// TIA Portal V19 export
DATA_BLOCK "DB_Panel_Posinfo"   // DB52
{ S7_Optimized_Access := 'FALSE' }
// stored: AutoNumber false
   VAR RETAIN
      Offset : Int := 50;   // * Beginn Daten
      Leng : Int := 80;   // * Länge Daten
      resDW1 : DWord := 16#0000_0000;
      resDW2 : DWord := 16#0000_0000;
      resDW3 : DWord := 16#0000_0000;
      resDW4 : DWord := 16#0000_0000;
      last_Takt : DInt := 0;
      Taktzeit : DInt := 0;   // Zeit die der Takt läuft
      Takt_Ware : DInt := 0;   // Zeit seit Ausfahrt letzte Fertigware
      Stop_Anlage : Byte := 16#00;   // ungleich 0-->Kettenbearbeitung anhalten
      Feierabend : Byte := 16#00;   // ungleich 0-->FEIERABENDPROGRAMM
      Sonder_BA : Byte := 16#00;   // ungleich 0-->ELEKTROLYSE, ENTMETALLISIEREN
      IST_Sonder_BA : Byte := 16#00;
      FB_FW_akt : Word := 16#0000;   // an Fernbedienung gewählter FW
      SPS_getaktet : Bool := TRUE;
      resDW10 : DWord := 16#0000_0000;
      resDW11 : DWord := 16#0000_0000;
      resW : Word := 16#0000;
      Pos : Array[1..30] of Struct   // * Feldlänge anpassen
         Prio_Pos : Byte;   // Priorität des Bades (höchste Priorität==0
         lngsm_IN : Bool;   // langsames Einsetzen erforderlich-abhängig von immer_schnell
         lngsm_OUT : Bool;   // langsames Ausheben erforderlich-abhängig von immer_schnell
         res : Bool;
         res1 : Bool;
         res2 : Bool;
         res3 : Bool;
         Luft_Ein : Bool;   // Lufteinblasung ein
         Luft_Auto : Bool;   // Lufteinblasung Automatik
         Verweilzeit : DInt;   // Verweilzeit
         KF_A : Real;   // Korrekturfaktor WT_Auslastung 0..100%-->0..1, Gesamtoberfläche
         KF_Expo : Real;   // Korrekturfaktor Expozeit in %
         T_Vorruf : Int;   // Vorrufzeit lößt Vorruf n Sekunden vor Ablauf der Expozeit aus
         T_Pend : Int;   // Auspendelzeit 0..999s
         T_ATZ : Int;   // Abtropfzeit 0..999s
         NS_Auto : Bool;   // Nachspeisung Automatik
         SR_Auto : Bool;   // Spritzregister Automatik
         res6 : Bool;
         WBE_Ein : Bool;   // Warenbewegung ein
         WBE_Auto : Bool;   // Warenbewegung Automatik
         TS_Pos : Bool;   // Tropfschalenpos.
         res9 : Bool;
         res10 : Bool;
         resB : Byte;
         Niv_SPR : Int;   // Stärke Spritzen
         Zeit_SPR : Int;   // Zeit Spritzen
         Niv_Luft : Int;   // Stärke Lufteinblasung
         Zeit_Luft : Int;   // Zeit Lufteinblasung
         Niv_NS : Int;   // Niveau Füllstand in %
         Zeit_NS : Int;   // Nachspeisezeit getaktete NS
         NS_Kor_Tr : Byte;   // Korrektur Nachspeisezeit für Trommel
         Coun_Kor : Byte;   // Counter Korrektur Nachspeisung
         resD : DInt;
         resR_1 : Real;
         resR_2 : Real;
         resR_3 : Real;
         resI_1 : Int;
         resI_2 : Int;
         ExpoTol : DInt;   // Toleranz Expozeit
         SonDW1 : DInt;   // freie Nutzung Gesamtzeit Rüttler
         SonDW2 : DInt;   // freie Nutzung Intervall ein Rüttler
         SonDW3 : DInt;   // freie Nutzung Intervall aus Rüttler
         SonDW4 : DInt;   // freie Nutzung (Verzögerung US-Rüttler)
         T_Zt_SR : Int;   // Test-Zeit Spritzregister
         T_Zt_NS : Int;   // Test-Zeit Nachspeisung
      END_STRUCT;
   END_VAR
BEGIN
   Pos[1..9].Prio_Pos := 16#05;
   Pos[10].Prio_Pos := 16#00;
   Pos[11..12].Prio_Pos := 16#01;
   Pos[13..14].Prio_Pos := 16#00;
   Pos[15..16].Prio_Pos := 16#01;
   Pos[17].Prio_Pos := 16#00;
   Pos[18].Prio_Pos := 16#01;
   Pos[19].Prio_Pos := 16#00;
   Pos[20..21].Prio_Pos := 16#01;
   Pos[22].Prio_Pos := 16#00;
   Pos[23].Prio_Pos := 16#02;
   Pos[24..27].Prio_Pos := 16#05;
   Pos[28].Prio_Pos := 16#02;
   Pos[29].Prio_Pos := 16#03;
   Pos[30].Prio_Pos := 16#02;
   Pos[1..30].lngsm_IN := FALSE;
   Pos[1..30].lngsm_OUT := FALSE;
   Pos[1..30].res := FALSE;
   Pos[1..30].res1 := FALSE;
   Pos[1..30].res2 := FALSE;
   Pos[1..30].res3 := FALSE;
   Pos[1..30].Luft_Ein := FALSE;
   Pos[1..30].Luft_Auto := FALSE;
   Pos[1].Verweilzeit := 0;
   Pos[2].Verweilzeit := 2107;
   Pos[3].Verweilzeit := 2074;
   Pos[4].Verweilzeit := 0;
   Pos[5].Verweilzeit := 32100;
   Pos[6..7].Verweilzeit := 0;
   Pos[8].Verweilzeit := 115;
   Pos[9..23].Verweilzeit := 0;
   Pos[24].Verweilzeit := 300;
   Pos[25..27].Verweilzeit := 0;
   Pos[28].Verweilzeit := 32;
   Pos[29].Verweilzeit := 1;
   Pos[30].Verweilzeit := 0;
   Pos[1..30].KF_A := 1000.0;
   Pos[1..30].KF_Expo := 1.0;
   Pos[1..30].T_Vorruf := 0;
   Pos[1..30].T_Pend := 1;
   Pos[1..2].T_ATZ := 0;
   Pos[3..7].T_ATZ := 10;
   Pos[8..9].T_ATZ := 5;
   Pos[10].T_ATZ := 10;
   Pos[11..12].T_ATZ := 5;
   Pos[13..14].T_ATZ := 10;
   Pos[15..16].T_ATZ := 5;
   Pos[17].T_ATZ := 10;
   Pos[18].T_ATZ := 5;
   Pos[19].T_ATZ := 10;
   Pos[20..21].T_ATZ := 5;
   Pos[22].T_ATZ := 10;
   Pos[23].T_ATZ := 5;
   Pos[24..27].T_ATZ := 2;
   Pos[28].T_ATZ := 0;
   Pos[29].T_ATZ := 5;
   Pos[30].T_ATZ := 2;
   Pos[1..30].NS_Auto := FALSE;
   Pos[1..25].SR_Auto := FALSE;
   Pos[26].SR_Auto := TRUE;
   Pos[27..29].SR_Auto := FALSE;
   Pos[30].SR_Auto := TRUE;
   Pos[1..30].res6 := FALSE;
   Pos[1..30].WBE_Ein := FALSE;
   Pos[1..30].WBE_Auto := FALSE;
   Pos[1..30].TS_Pos := FALSE;
   Pos[1..30].res9 := FALSE;
   Pos[1..30].res10 := FALSE;
   Pos[1..30].resB := 16#00;
   Pos[1..30].Niv_SPR := 0;
   Pos[1..30].Zeit_SPR := 0;
   Pos[1..30].Niv_Luft := 0;
   Pos[1..30].Zeit_Luft := 0;
   Pos[1..30].Niv_NS := 0;
   Pos[1..30].Zeit_NS := 0;
   Pos[1..30].NS_Kor_Tr := 16#00;
   Pos[1..30].Coun_Kor := 16#00;
   Pos[1..30].resD := 0;
   Pos[1..30].resR_1 := 0.0;
   Pos[1..30].resR_2 := 0.0;
   Pos[1..30].resR_3 := 0.0;
   Pos[1..30].resI_1 := 0;
   Pos[1..30].resI_2 := 0;
   Pos[1..9].ExpoTol := 600;
   Pos[10..22].ExpoTol := 0;
   Pos[23..27].ExpoTol := 600;
   Pos[28..30].ExpoTol := 60;
   Pos[1..30].SonDW1 := 0;
   Pos[1..30].SonDW2 := 0;
   Pos[1..30].SonDW3 := 0;
   Pos[1..30].SonDW4 := 0;
   Pos[1..30].T_Zt_SR := 0;
   Pos[1..30].T_Zt_NS := 0;
END_DATA_BLOCK
